FUNCTION_BLOCK FoldingMachine
VAR_INPUT
	//enable AT %Q* : BOOL;
	//reset AT %Q* : BOOL;
	foldingPositions AT %Q* : ARRAY[0..1] OF INT;
	
	lifterExtend AT %Q* : BOOL;
	lifterHalf AT %Q* : BOOL;
	lifterRetract AT %Q* : BOOL;
	
	benderExtend AT %Q* : BOOL;
	benderRetract AT %Q* : BOOL;
END_VAR
VAR_OUTPUT
	activeMaterial : STRING;
	
	lifterExtended AT %I* : BOOL;
	lifterIntermediate AT %I* : BOOL;
	lifterRetracted AT %I* : BOOL;
	
	benderExtended AT %I* : BOOL;
	benderRetracted AT %I* : BOOL;
	
	suction : SuctionPad;
	
	occupied AT %I* : BOOL;
	manifoldOk AT %I* : BOOL;
	
	//ready AT %I* : BOOL;
	//busy AT %I* : BOOL;
	//done AT %I* : BOOL;	
END_VAR

METHOD setFoldingPositions : BOOL
VAR_INPUT
	foldPos0, foldPos1 : INT;
END_VAR
foldingPositions[0] := foldPos0;
foldingPositions[1] := foldPos1;
END_METHOD

END_FUNCTION_BLOCK

(* stored: Version 1.1.0.1, ProductVersion 3.1.4024.11
   POU FoldingMachine: Id {d6ca17f9-19c5-43ef-9652-b5b02a8cedeb}, SpecialFunc None
   Method setFoldingPositions: Id {0c92faf8-7c73-471c-9944-f27c4a400706} *)
